{attribute 'qualified_only'}
VAR_GLOBAL
	bBuildGroup	: BOOL;
	bLoad		: BOOL;
	bStart		: BOOL;
	bStop		: BOOL;
	bReset		: BOOL;
END_VAR

(* stored: Version 1.1.0.1, ProductVersion 3.1.4024.2
   GVL gcode: Id {f58b9562-53a1-4d3c-a228-3a03bf0660ef} *)
